ABB RAPID module: TCP_t2B2.MOD

MODULE TCP_t2B2
	! Points are read in order of declaration.
  ! Please do not change the order of points!

  LOCAL PERS robtarget pTCP_Point1:=[[515.4955,32.57635,293.049],[0.511388003826141,0.330361515283585,0.781470715999603,-0.136554583907127],[0,-2,1,0],[9E+09,9E+09,9E+09,9E+09,9E+09,9E+09]];
	LOCAL PERS robtarget pTCP_Point2:=[[512.8115,-19.87533,296.8105],[0.518410265445709,-0.0439002774655819,0.851206660270691,0.0690709128975868],[-1,1,-2,0],[9E+09,9E+09,9E+09,9E+09,9E+09,9E+09]];
	LOCAL PERS robtarget pTCP_Point3:=[[545.7906,13.85153,310.3502],[0.285668164491653,-0.393444567918777,0.873814761638641,-0.0065390202216804],[-1,0,-2,0],[9E+09,9E+09,9E+09,9E+09,9E+09,9E+09]];
	LOCAL PERS robtarget pTCP_Point4:=[[623.4874,-19.87568,298.1783],[0.0294857658445835,0.0928741246461868,-0.987644195556641,-0.122735239565372],[-1,0,-1,0],[9E+09,9E+09,9E+09,9E+09,9E+09,9E+09]];

ENDMODULE
